// TIA Portal V16 export
// export: Created 2022-02-11T14:39:21.3631075Z, ExportSetting WithDefaults, DisplayName Totally Integrated Automation Portal, DisplayVersion V16 Update 1, DisplayName TIA Portal Version Control Interface, DisplayVersion V16, DisplayName TIA Portal Openness, DisplayVersion V16, DisplayName SINAMICS Startdrive Advanced, DisplayVersion V16 Update 5, DisplayName SINAMICS Startdrive G130, G150, S120, S150, SINAMICS MV, S210, DisplayVersion V16 Update 5, DisplayName SINAMICS Startdrive G110M, G120, G120C, G120D, G120P, G115D, DisplayVersion V16 Update 5, DisplayName STEP 7 Professional, DisplayVersion V16, DisplayName STEP 7 Safety, DisplayVersion V16, DisplayName WinCC Advanced, DisplayVersion V16, DisplayName SIMATIC Visualization Architect, DisplayVersion V16
DATA_BLOCK "Безопасность_DB"   // DB1
VERSION : 0.1
// stored: AutoNumber true, InstanceOfName Безопасность, InstanceOfType FB
"Безопасность"
   // VAR RETAIN
   //    Trig61 : Bool;
   //    Trig62 : Bool;
   //    Trig63 : Bool;
   //    Trig64 : Bool;
   //    Trig65 : Bool;
   //    Trig66 : Bool;
   //    Trig67 : Bool;
   //    Trig69 : Bool;
   //    Trig68 : Bool;
   //    ProhibitionLoading : Bool;
   //    ProhibitionDefect : Bool;
   //    ProhibitionSorting : Bool;
   //    ProhibitionGasket : Bool;
   // END_VAR
BEGIN
END_DATA_BLOCK
